FUNCTION_BLOCK MS_model
  (* Version 1.0, 2005-09-20, Goran Cengic, Chalmers *)
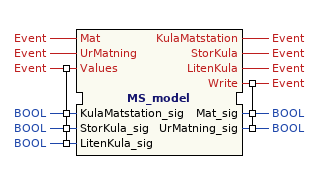
  EVENT_INPUT
    Mat;
    UrMatning;
    Values WITH KulaMatstation_sig, StorKula_sig, LitenKula_sig;
  END_EVENT
  EVENT_OUTPUT
    KulaMatstation;
    StorKula;
    LitenKula;
    Write WITH Mat_sig, UrMatning_sig;
  END_EVENT
  VAR_INPUT
    KulaMatstation_sig : BOOL;
    StorKula_sig : BOOL;
    LitenKula_sig : BOOL;
  END_VAR
  VAR_OUTPUT
    Mat_sig : BOOL;
    UrMatning_sig : BOOL;
  END_VAR
  VAR
    StorKula_var : BOOL;
    LitenKula_var : BOOL;
  END_VAR
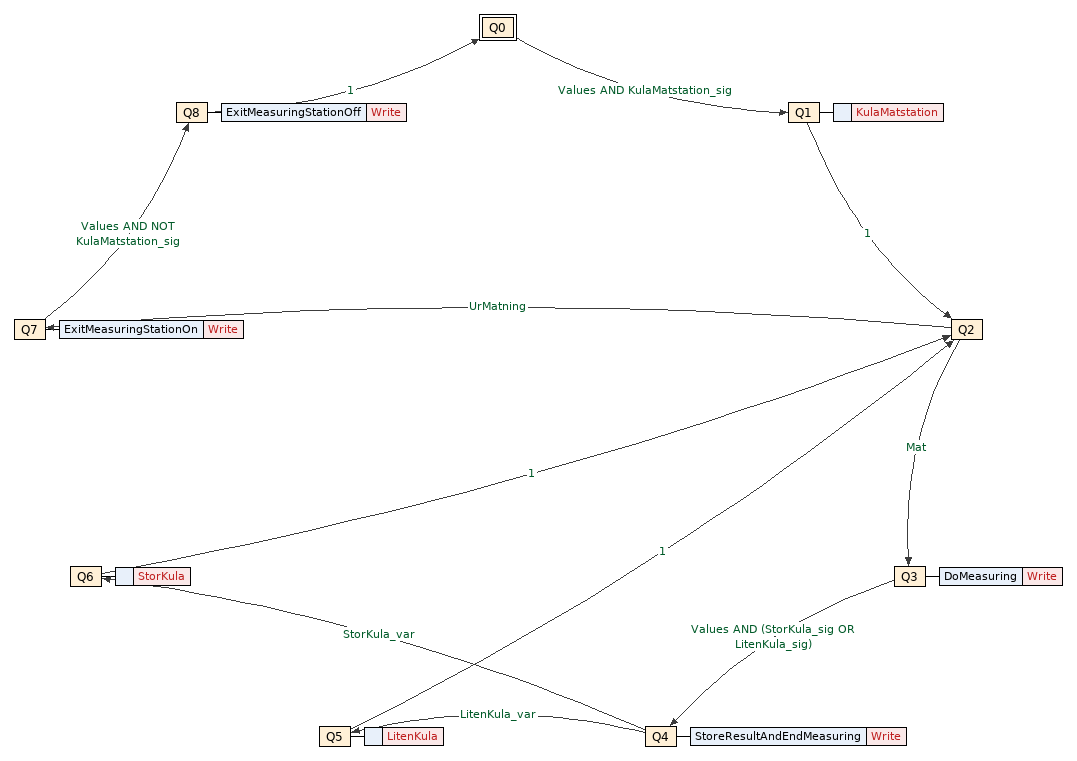
  EC_STATES
    Q0;
    Q1 : -> KulaMatstation;
    Q2;
    Q3 : DoMeasuring -> Write;
    Q4 : StoreResultAndEndMeasuring -> Write;
    Q5 : -> LitenKula;
    Q6 : -> StorKula;
    Q7 : ExitMeasuringStationOn -> Write;
    Q8 : ExitMeasuringStationOff -> Write;
  END_STATES
  EC_TRANSITIONS
    Q0 TO Q1 := Values AND KulaMatstation_sig;
    Q1 TO Q2 := 1;
    Q2 TO Q3 := Mat;
    Q2 TO Q7 := UrMatning;
    Q3 TO Q4 := Values AND (StorKula_sig OR LitenKula_sig);
    Q4 TO Q5 := LitenKula_var;
    Q4 TO Q6 := StorKula_var;
    Q5 TO Q2 := 1;
    Q6 TO Q2 := 1;
    Q7 TO Q8 := Values AND NOT KulaMatstation_sig;
    Q8 TO Q0 := 1;
  END_TRANSITIONS
  ALGORITHM DoMeasuring IN Java:
		System.out.println("Start measuring.");
		Mat_sig = true;
  END_ALGORITHM
  ALGORITHM StoreResultAndEndMeasuring IN Java:
		System.out.println("Store result and end measuring.");
		StorKula_var = StorKula_sig;
		LitenKula_var = LitenKula_sig;
		System.out.println("StorKula=" + StorKula_var + " LitenKula=" + LitenKula_var);
		Mat_sig = false;
  END_ALGORITHM
  ALGORITHM ExitMeasuringStationOn IN Java:
		System.out.println("Exit measuring station ON.");
		UrMatning_sig = true;
  END_ALGORITHM
  ALGORITHM ExitMeasuringStationOff IN Java:
		System.out.println("Exit measuring station OFF.");
		UrMatning_sig = false;
  END_ALGORITHM
END_FUNCTION_BLOCK
